// TIA Portal V20 export
ORGANIZATION_BLOCK "Main"   // OB1, LAD, ProgramCycle
TITLE = "Main Program Sweep (Cycle)"
{ S7_Optimized_Access := 'TRUE' }
// stored: SetENOAutomatically false
   VAR_INPUT
      Initial_Call : Bool;   // Initial call of this OB
      Remanence : Bool;   // =True, if remanent data are available
   END_VAR
BEGIN

REGION Network 1
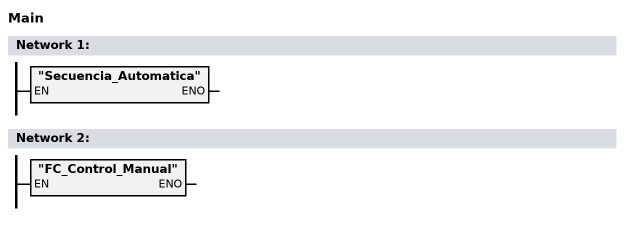
   RUNG wire#powerrail
      "Secuencia_Automatica"()
   END_RUNG
   // the same network as SCL:
   "Secuencia_Automatica"();
END_REGION

REGION Network 2
   RUNG wire#powerrail
      "FC_Control_Manual"()
   END_RUNG
   // the same network as SCL:
   "FC_Control_Manual"();
END_REGION
END_ORGANIZATION_BLOCK
